// TwinCAT 3 PLC project PLC
// ProgramVersion: 3.1.4024.0
// libraries:
//   Tc2_Standard, * (Beckhoff Automation GmbH)
//   Tc2_System, * (Beckhoff Automation GmbH)
//   Tc3_Module, * (Beckhoff Automation GmbH)
// project tree:
//   / PlcTask.TcTTO
//   POUs/ FBD.TcPOU, LLD.TcPOU, MAIN.TcPOU, SFC.TcPOU
// real-time tasks:
//   TASK PlcTask: cycle T#10ms, priority 20, ADS port 350

CONFIGURATION PLC
    RESOURCE PLC ON TwinCAT3
        TASK PlcTask(INTERVAL := T#10ms, PRIORITY := 20);
        PROGRAM MAIN WITH PlcTask : MAIN;
    END_RESOURCE
END_CONFIGURATION

// ---- POUs/MAIN.TcPOU
PROGRAM MAIN
VAR
END_VAR

FBD();

END_PROGRAM

// ---- POUs/FBD.TcPOU
PROGRAM FBD
VAR
	count : INT := 0;
	reset : BOOL := FALSE;
END_VAR

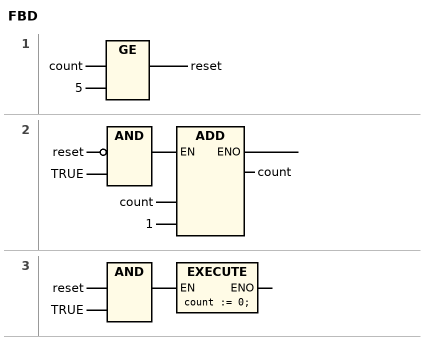
// NETWORK 1
reset := count >= 5;

// NETWORK 2
IF NOT reset AND TRUE THEN count := count + 1; END_IF

// NETWORK 3
IF reset AND TRUE THEN count := 0; END_IF

END_PROGRAM

// ---- POUs/LLD.TcPOU
PROGRAM LLD
VAR
	count : INT := 0;
	reset : BOOL := FALSE;
	
END_VAR
VAR // added by the converter: edge detectors and wires of the graphical bodies
    _w1, _w2 : BOOL;
END_VAR

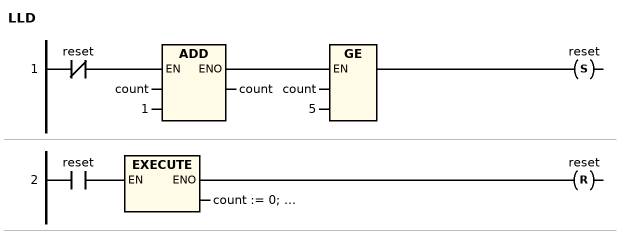
// NETWORK 1
_w1 := NOT reset;
IF _w1 THEN count := count + 1; END_IF
reset S= _w1 AND count >= 5;

// NETWORK 2
_w2 := reset;
IF _w2 THEN count := 0; END_IF
reset R= _w2;

END_PROGRAM

// ---- POUs/SFC.TcPOU
PROGRAM SFC
VAR
	count : INT := 0;
	reset : BOOL := FALSE;
END_VAR

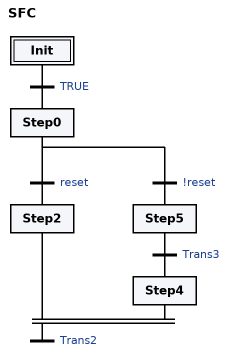
INITIAL_STEP Init:
END_STEP
TRANSITION FROM Init TO Step0
    := TRUE;
END_TRANSITION
STEP Step0:
END_STEP
TRANSITION FROM Step0 TO Step2
    := reset;
END_TRANSITION
STEP Step2:
END_STEP
TRANSITION FROM Step0 TO Step5
    := !reset;
END_TRANSITION
STEP Step5:
END_STEP
TRANSITION FROM Step5 TO Step4
    := Trans3;
END_TRANSITION
STEP Step4:
END_STEP
TRANSITION FROM (Step2, Step4) TO ???
    := Trans2;
END_TRANSITION

ACTION Step5_entry:
count := count + 1;
END_ACTION

END_PROGRAM
